{attribute 'pack_mode' := '1'}
TYPE OutgoingMessage :
STRUCT
	version: LINT; (* Matches the serialVersionUID of the equivalent Java class.*)
END_STRUCT
END_TYPE

(* stored: Version 1.1.0.1, ProductVersion 3.1.4022.12
   DUT OutgoingMessage: Id {33a5b42b-aebc-4eb1-9adf-b18031df431f} *)
